TYPE (* logiBUS DI Struct Dual *)
  (* Version 1.0, 2026-05-28, franz *)
  PACKAGE logiBUS::io::DI;
  logiBUS_DI_S_Dual : STRUCT
    Up : logiBUS::io::DI::logiBUS_DI_S := (Pin := 255); (* forward, up, right, clockwise *)
    Down : logiBUS::io::DI::logiBUS_DI_S := (Pin := 255); (* backward, down, left, counter-clockwise *)
  END_STRUCT;
END_TYPE
